TYPE E_GasType :
(
    none := 0,
    Nitrogen,
    Argon
);
END_TYPE

(* stored: Version 1.1.0.1, ProductVersion 3.1.4022.18
   DUT E_GasType: Id {e6f93326-faf5-4939-952f-051eed70a044} *)
